// Mitsubishi GX Works2 project: RollerConveyor   PLC: Q03UD

PROGRAM MAIN
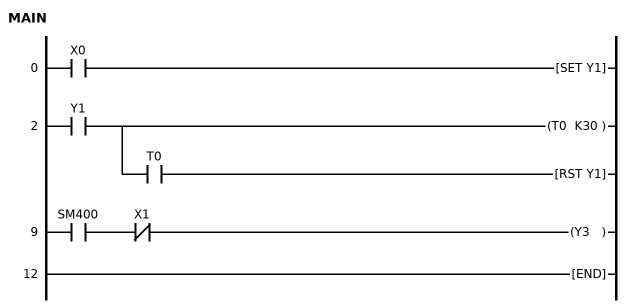
0     LD      X0
      SET     Y1
2     LD      Y1
      OUT     T0 K30
      AND     T0
      RST     Y1
9     LD      SM400
      ANI     X1
      OUT     Y3
12    END
END_PROGRAM
